// TIA Portal V17 export
// export: Created 2025-03-07T09:16:34.3206185Z, ExportSetting WithDefaults, DisplayName Totally Integrated Automation Portal, DisplayVersion V17 Update 8, DisplayName TIA Portal Openness, DisplayVersion V17 Update 8, DisplayName TIA Portal Version Control Interface, DisplayVersion V17, DisplayName SINAMICS Startdrive Advanced, DisplayVersion V17 SP2, DisplayName SINAMICS Startdrive G110M, G120, G120C, G120D, G120P, G115D, DisplayVersion V17 SP2, DisplayName SINAMICS Startdrive G130, G150, S120, S150, SINAMICS MV, S210, DisplayVersion V17 SP2, DisplayName STEP 7 Professional, DisplayVersion V17 Update 8, DisplayName SINUMERIK ONE STEP 7 Toolbox, DisplayVersion V17 Update 12, DisplayName SINUMERIK 840D sl STEP 7 Toolbox, DisplayVersion V17 Update 12, DisplayName STEP 7 Safety, DisplayVersion V17 Update 6, DisplayName WinCC Advanced, DisplayVersion V17 Update 8
DATA_BLOCK "LBP_TMTurretMT"   // DB1073
TITLE = Tool management / Gestión de herramientas / Werkzeugverwaltung
{ S7_Optimized_Access := 'FALSE'; DB_Accessible_From_OPC_UA := 'FALSE' }
AUTHOR : SINUMERIK
FAMILY : SINUMERIK_ONE
VERSION : 6.15
// Interface between user program and tool management, contains signals for turret (multitool). / Interfaz entre programa de usuario y gestión de herramientas, contiene señales para torreta/revólver (Multitool). / Schnittstelle zwischen Anwenderprogramm und Werkzeugverwaltung, enthält Signale für Revolver (Multitool)
// stored: AutoNumber false, DBAccessibleFromOPCUA false, DBAccessibleFromWebserver true, InstanceOfName LBP_typeTMTurretMT, InstanceOfType UDT, IsOnlyStoredInLoadMemory false, IsWriteProtectedInAS false
"LBP_typeTMTurretMT"
   // VAR RETAIN
   //    MTIF : Array[1..16] of Struct
   //       DistanceCoding : Int;
   //       Places : Int;
   //       Distance : Real;
   //       NewMTNo : Int;
   //       NewPlace : Int;
   //       OldMTNo : Int;
   //       OldPlace : Int;
   //       LocType : Int;
   //       SLeft : Int;
   //       SRight : Int;
   //       STop : Int;
   //       SBottom : Int;
   //       TInBuffer : Bool;
   //       IgnoreDisabled : Bool;
   //       Unload : Bool;
   //       Load : Bool;
   //       MasterTool : Bool;
   //       n26_5 : Bool;
   //       n26_6 : Bool;
   //       HandTool : Bool;
   //       Active : Bool;
   //       Enabled : Bool;
   //       Disabled : Bool;
   //       Measured : Bool;
   //       Prewarn : Bool;
   //       Change : Bool;
   //       FixedLoc : Bool;
   //       Used : Bool;
   //       TNo : Int;
   //       Toolholder : Int;
   //       MyMag : Int;
   //       MyPlace : Int;
   //       reserved : Array[1..7] of Int;
   //    END_STRUCT;
   // END_VAR
BEGIN
END_DATA_BLOCK
